# EPICS substitutions: elioApp/Db/EL2124.substitutions
file EL2124.template { pattern
{ CHAN	}
{ 1	}
{ 2	}
{ 3	}
{ 4	}
}
